FUNCTION_BLOCK FB_Torque_prediction
VAR_INPUT
	Lh_depth:REAL;
	Rh_depth:REAL;
	Levels:ARRAY[0..31]OF REAL;
	Bottom_level:REAL;
	Enable:BOOL;
	Lh_full_load:BOOL;
	Lh_half_load:BOOL;
	Rh_full_load:BOOL;
	Rh_half_load:BOOL;
	Speed_ref:REAL;
	Speed:REAL;
	Speed_control:BOOL;
END_VAR
VAR_OUTPUT
	Predicted_current:REAL;
END_VAR
VAR
	Speed_ref_prev:REAL;
	Speed_ramp_rate:REAL;
	Moving_fwd:BOOL;
	Moving_rev:BOOL;
	Rev_pulse:BOOL;
	Fwd_pulse:BOOL;
	FB_LAG_FILTER_0: FB_Lag_filter;
	RS_0: RS;
	RS_1: RS;
	FB_TP_with_stop_0: FB_TP_with_stop;
	FB_TP_with_stop_1: FB_TP_with_stop;
END_VAR

M_Torque_prediction();

END_FUNCTION_BLOCK

(* stored: Version 1.1.0.1, ProductVersion 3.1.4024.0
   POU FB_Torque_prediction: Id {f9827b8e-6bb8-46fa-b7c6-ace3b65a6f4d}, SpecialFunc None *)
